// TIA Portal project "一个按钮控制两台电机模拟" (V15.1)

(* hardware
DEVICE "S7-1200 station_1"  S7-1200 Station
   slot 0: "Rack_0"  S7-1200 Rack  Rack  V1.0
   slot 1: "PLC_1"  CPU 1212C DC/DC/DC  6ES7 212-1AE40-0XB0  V4.2
*)

// ===== PLC "PLC_1"  CPU 1212C DC/DC/DC =====

VAR_GLOBAL   // PLC tag table "默认变量表"
   ""启动"" AT %I0.0 : Bool;
   ""停止"" AT %I0.1 : Bool;
   ""开启"" AT %I0.4 : Bool;
   ""电机"" AT %Q0.0 : Bool;
   ""电机1"" AT %Q0.4 : Bool;
   ""电机2"" AT %Q0.5 : Bool;
END_VAR